(* IEC 61131-3 sources: TwinCATProj/TwinCATRD/PPS_Archive_fb/Functions/PPSFun, 11 files *)

(* ---- PPSFun.typ ---- *)
(********************************************************************
 * COPYRIGHT -- Pro Pack Systems, Inc.
 ********************************************************************
 * Library: PPSFun
 * File: PPSFun.typ
 * Author: Paul Zurlinden
 * Created: November 03, 2010
 ********************************************************************
 * Data types of library PPSFun
 ********************************************************************)

TYPE
	dtEasyLight_Outputs : 	STRUCT
		xCmdActive : BOOL;
		diResult : DINT;
		sResultText : STRING[41];
	END_STRUCT;
	dtEasyLight_InputOutput : 	STRUCT
		diCmd : DINT;
	END_STRUCT;
	dtEasyLightInterface : 	STRUCT
		Q : dtEasyLight_Outputs;
		IQ : dtEasyLight_InputOutput;
	END_STRUCT;
	dtVacCupInputs : 	STRUCT
		xEnable : BOOL;
		xEnManCntrl : BOOL;
		xManCmd : BOOL;
		tPurgeTime : TIME;
		xEmergency : BOOL;
	END_STRUCT;
	dtVacCupInputs2 : 	STRUCT
		xEnable : BOOL;
		xEnManCntrl : BOOL;
		xManCmd : BOOL;
		tPurgeTime : TIME;
		xEmergency : BOOL;
		sName : STRING[40];
		xMonitored : BOOL;
		tMonitorDelay : TIME;
	END_STRUCT;
	dtVacCup_InOut2 : 	STRUCT
		xAutoOn : BOOL;
		xAutoOff : BOOL;
		xClearFault : BOOL;
	END_STRUCT;
	dtVacCup_InOut : 	STRUCT
		xAutoOn : BOOL;
		xAutoOff : BOOL;
	END_STRUCT;
	dtVacCupOuputs : 	STRUCT
		xFBActive : BOOL;
		xSVPurge : BOOL;
		xSVVac : BOOL;
	END_STRUCT;
	dtVacCupOuputs2 : 	STRUCT
		xFBActive : BOOL;
		xSVPurge : BOOL;
		xSVVac : BOOL;
		xFault : BOOL;
		sFaultTxt : STRING[82];
	END_STRUCT;
	dtVacuumCupInterface : 	STRUCT
		I : dtVacCupInputs;
		IQ : dtVacCup_InOut;
		Q : dtVacCupOuputs;
	END_STRUCT;
	dtVacuumCupInterface2 : 	STRUCT
		I : dtVacCupInputs2;
		IQ : dtVacCup_InOut2;
		Monitor : dtDebounceInterface;
		Q : dtVacCupOuputs2;
		stErrData : dtFB_ErrorData;
	END_STRUCT;
	EnumerationEasyLight :
		(
		EN_EZL_GNSteady := 1,
		EN_EZL_RDSteady := 2,
		EN_EZL_YWSteady := 3,
		EN_EZL_BUSteady := 4,
		EN_EZL_GNFlash := 5,
		EN_EZL_RDFlash := 6,
		EN_EZL_YWFlash := 7,
		EN_EZL_BUFlash := 8,
		EN_EZL_AltGnRd := 9,
		EN_EZL_AltRdBu := 10,
		EN_EZL_AltGnYw := 11,
		EN_EZL_AltGnBu := 12,
		EN_EZL_AltRdYw := 13,
		EN_EZL_AltYwBu := 14,
		EN_EZL_AltGnRdYwBu := 15,
		EN_EZL_AllOff := 16
		);
	dtGlueApplictor : 	STRUCT
		xEnable : BOOL;
		xApplyCmd : BOOL;
		xEnManual : BOOL;
		xManPurgeCmd : BOOL;
		tPurgeTime : TIME;
		xEmergency : BOOL;
	END_STRUCT;
	dtDigCntrlInterface : 	STRUCT
		I : dtDigCntrl_Inputs;
		IQ : dtDigCntrl_InOut;
		Q : dtDigCntrl_Outputs;
		stMonitor : dtDebounceInterface;
		stErrData : dtFB_ErrorData;
	END_STRUCT;
	dtDigCntrl_Inputs : 	STRUCT
		xEnManCntrl : BOOL;
		xManCmd : BOOL;
		xEmergency : BOOL;
		xEnMonitor : BOOL;
		tMonitorDelay : TIME;
	END_STRUCT;
	dtDigCntrl_InOut : 	STRUCT
		xAutoOn : BOOL;
		xAutoOff : BOOL;
		xFaultReset : BOOL;
	END_STRUCT;
	dtDigCntrl_Outputs : 	STRUCT
		xCmd : BOOL;
		xFault : BOOL;
	END_STRUCT;
	dtFB_ErrorData : 	STRUCT
		uiErrorID : UINT;
		sErrorString : STRING[80];
		sSourceName : STRING[80];
	END_STRUCT;
	dtDebounceInterface : 	STRUCT
		I : dtDebounce_Inputs;
		Q : dtDebounce_Outputs;
	END_STRUCT;
	dtDebounce_Inputs : 	STRUCT
		xSignal : BOOL;
		tOnDelay : TIME;
		tOffDelay : TIME;
	END_STRUCT;
	dtDebounce_Outputs : 	STRUCT
		xCmd : BOOL;
		tOnTimer : TIME;
		tOffTimer : TIME;
	END_STRUCT;
	dtCylCntrlInterface : 	STRUCT
		I : dtCylCntrl_Inputs;
		IQ : dtCylCntrl_InOut;
		Q : dtCylCntrl_Outputs;
		stSensorExt : dtDebounceInterface;
		stSensorRet : dtDebounceInterface;
	END_STRUCT;
	dtCylCntrl_Inputs : 	STRUCT
		xEnableFB : BOOL;
		xValveOffRetract : BOOL;
		xAirOk : BOOL;
		xEnManCntrl : BOOL;
		xManCmd : BOOL;
		xEmergency : BOOL;
		xEnMonitor : BOOL;
		usiHWFamily : USINT;
		tTravelDel : TIME;
		xFaultReset : BOOL;
	END_STRUCT;
	dtCylCntrl_InOut : 	STRUCT
		xExtCmd : BOOL;
		xRetCmd : BOOL;
	END_STRUCT;
	dtCylCntrl_Outputs : 	STRUCT
		xFBActive : BOOL;
		xSVCmd : BOOL;
		xExtended : BOOL;
		xRetracted : BOOL;
		xFaultNoExt : BOOL;
		xFaultNoRet : BOOL;
	END_STRUCT;
END_TYPE

(* ---- FB_CylCntrl.st ---- *)
(********************************************************************
 * COPYRIGHT -- Pro Pack Systems, Inc.
 ********************************************************************
 * Library: PPSFun
 * File: FB_CylCntrl.st
 * Author: Paul Zurlinden
 * Created: November 04, 2010
 ********************************************************************
 * Implementation of library PPSFun
 ********************************************************************)

(* Controls a pneumatic cylinder with or without end of travel sensors *)
FUNCTION_BLOCK FB_CylCntrl

Timer(PT := iq_CylCntrlInterface.I.tTravelDel);
RT(CLK := iq_CylCntrlInterface.I.xManCmd);
RT_Air(CLK := iq_CylCntrlInterface.I.xAirOk);

(* Debounce Cylinder Position Sensors *)
IF iq_CylCntrlInterface.I.xEnMonitor THEN
	aFB_SensExt[0](iq_DebounceInterface := iq_CylCntrlInterface.stSensorExt);
	aFB_SensExt[1](iq_DebounceInterface := iq_CylCntrlInterface.stSensorRet);
END_IF

IF iq_CylCntrlInterface.Q.xFaultNoExt OR iq_CylCntrlInterface.Q.xFaultNoRet THEN
	xFaultSum := TRUE;
ELSE
	xFaultSum	:= FALSE;
END_IF

IF iq_CylCntrlInterface.I.xFaultReset THEN
	iq_CylCntrlInterface.Q.xFaultNoExt	:= FALSE;
	iq_CylCntrlInterface.Q.xFaultNoRet := FALSE;
END_IF

IF iq_CylCntrlInterface.I.xEnableFB THEN
	iq_CylCntrlInterface.Q.xFBActive	:= TRUE;

	(* Determine Cylinder Position when air is first turned on *)
	IF RT_Air.Q THEN
		IF iq_CylCntrlInterface.I.xEnMonitor THEN
	 		IF iq_CylCntrlInterface.stSensorExt.Q.xCmd THEN
  				iq_CylCntrlInterface.Q.xExtended		:= TRUE;
   			ELSIF iq_CylCntrlInterface.stSensorRet.Q.xCmd THEN
			 	iq_CylCntrlInterface.Q.xRetracted	:= TRUE;
   			END_IF
		ELSE
			IF iq_CylCntrlInterface.I.xValveOffRetract THEN
   				IF iq_CylCntrlInterface.Q.xSVCmd THEN
					iq_CylCntrlInterface.Q.xExtended := TRUE;
	 			ELSE
				   	iq_CylCntrlInterface.Q.xRetracted := TRUE;
	 			END_IF
			ELSE
				IF iq_CylCntrlInterface.Q.xSVCmd THEN
					iq_CylCntrlInterface.Q.xRetracted := TRUE;
	 			ELSE
				   	iq_CylCntrlInterface.Q.xExtended := TRUE;
	 			END_IF
			END_IF
		END_IF
	END_IF

	(* Fault monitor *)
	IF iq_CylCntrlInterface.I.xEnMonitor (*AND iq_CylCntrlInterface.I.usiHWFamily <> 4*) THEN (* Fault Monitor is enabled *)
		IF NOT xFaultSum THEN
			IF iq_CylCntrlInterface.I.xValveOffRetract THEN
				IF iq_CylCntrlInterface.Q.xSVCmd THEN
					IF iq_CylCntrlInterface.stSensorExt.Q.xCmd THEN
						iq_CylCntrlInterface.Q.xExtended			:= TRUE;
						iq_CylCntrlInterface.Q.xFaultNoExt		:= FALSE;
						Timer.IN												:= FALSE;
					ELSE
						IF Timer.Q THEN
							iq_CylCntrlInterface.Q.xExtended		:= FALSE;
							iq_CylCntrlInterface.Q.xFaultNoExt	:= TRUE;
							Timer.IN											:= FALSE;
						END_IF
					END_IF
				ELSE
					IF iq_CylCntrlInterface.stSensorRet.Q.xCmd THEN
						iq_CylCntrlInterface.Q.xRetracted 		:= TRUE;
						iq_CylCntrlInterface.Q.xFaultNoRet		:= FALSE;
						Timer.IN												:= FALSE;
					ELSE
						IF Timer.Q THEN
							iq_CylCntrlInterface.Q.xRetracted	:= FALSE;
							iq_CylCntrlInterface.Q.xFaultNoRet	:= TRUE;
							Timer.IN											:= FALSE;
						END_IF
					END_IF
				END_IF
			ELSE
				IF NOT iq_CylCntrlInterface.Q.xSVCmd THEN
					IF iq_CylCntrlInterface.stSensorExt.Q.xCmd THEN
						iq_CylCntrlInterface.Q.xExtended			:= TRUE;
						iq_CylCntrlInterface.Q.xFaultNoExt		:= FALSE;
						Timer.IN												:= FALSE;
					ELSE
						IF Timer.Q THEN
							iq_CylCntrlInterface.Q.xExtended		:= FALSE;
							iq_CylCntrlInterface.Q.xFaultNoExt	:= TRUE;
							Timer.IN	:= FALSE;
						END_IF
					END_IF
				ELSE
					IF iq_CylCntrlInterface.stSensorRet.Q.xCmd THEN
						iq_CylCntrlInterface.Q.xRetracted		:= TRUE;
						iq_CylCntrlInterface.Q.xFaultNoRet		:= FALSE;
						Timer.IN	:= FALSE;
					ELSE
						IF Timer.Q THEN
							iq_CylCntrlInterface.Q.xRetracted	:= FALSE;
							iq_CylCntrlInterface.Q.xFaultNoRet	:= TRUE;
							Timer.IN											:= FALSE;
						END_IF
					END_IF
				END_IF
			END_IF
		END_IF
	ELSE (* Fault Monitor is disabled *)
		IF iq_CylCntrlInterface.Q.xSVCmd THEN
			IF Timer.Q THEN
				IF iq_CylCntrlInterface.I.xValveOffRetract THEN
					iq_CylCntrlInterface.Q.xExtended		:= TRUE;
				ELSE
					iq_CylCntrlInterface.Q.xRetracted	:= TRUE;
				END_IF
				Timer.IN												:= FALSE;
			END_IF
		ELSE
			IF Timer.Q THEN
				IF iq_CylCntrlInterface.I.xValveOffRetract THEN
					iq_CylCntrlInterface.Q.xRetracted	:= TRUE;
				ELSE
					iq_CylCntrlInterface.Q.xExtended		:= TRUE;
	 			END_IF
				Timer.IN												:= FALSE;
			END_IF
		END_IF
	END_IF
	(* End Fault Monitor *)

	(* Control output *)
	IF iq_CylCntrlInterface.I.xEmergency OR xFaultSum THEN
		iq_CylCntrlInterface.Q.xSVCmd := FALSE;
	ELSE
		IF NOT iq_CylCntrlInterface.I.xEnManCntrl THEN (* When not in Manual Mode, control output *)

			IF iq_CylCntrlInterface.I.xValveOffRetract THEN
				IF iq_CylCntrlInterface.IQ.xExtCmd (*AND NOT iq_CylCntrlInterface.Q.xSVCmd*) THEN
					iq_CylCntrlInterface.Q.xSVCmd		:= TRUE;
					iq_CylCntrlInterface.Q.xRetracted	:= FALSE;
					iq_CylCntrlInterface.Q.xExtended		:= FALSE;
					Timer.IN											:= TRUE;
					IF iq_CylCntrlInterface.Q.xSVCmd THEN
						iq_CylCntrlInterface.IQ.xExtCmd		:= FALSE;
					END_IF
				END_IF

				IF iq_CylCntrlInterface.IQ.xRetCmd (*AND iq_CylCntrlInterface.Q.xSVCmd*) THEN
					iq_CylCntrlInterface.Q.xSVCmd		:= FALSE;
					iq_CylCntrlInterface.Q.xExtended		:= FALSE;
					iq_CylCntrlInterface.Q.xRetracted	:= FALSE;
					Timer.IN											:= TRUE;
					IF NOT iq_CylCntrlInterface.Q.xSVCmd THEN
						iq_CylCntrlInterface.IQ.xRetCmd		:= FALSE;
					END_IF
				END_IF
			ELSE
				IF iq_CylCntrlInterface.IQ.xExtCmd (*AND iq_CylCntrlInterface.Q.xSVCmd*) THEN
					iq_CylCntrlInterface.Q.xSVCmd		:= FALSE;
					iq_CylCntrlInterface.Q.xExtended		:= FALSE;
					iq_CylCntrlInterface.Q.xRetracted	:= FALSE;
					Timer.IN											:= TRUE;
					IF NOT iq_CylCntrlInterface.Q.xSVCmd THEN
						iq_CylCntrlInterface.IQ.xExtCmd		:= FALSE;
					END_IF
				END_IF

				IF iq_CylCntrlInterface.IQ.xRetCmd (*AND NOT iq_CylCntrlInterface.Q.xSVCmd*) THEN
					iq_CylCntrlInterface.Q.xSVCmd		:= TRUE;
					iq_CylCntrlInterface.Q.xExtended		:= FALSE;
					iq_CylCntrlInterface.Q.xRetracted	:= FALSE;
					Timer.IN											:= TRUE;
					IF iq_CylCntrlInterface.Q.xSVCmd THEN
						iq_CylCntrlInterface.IQ.xRetCmd		:= FALSE;
					END_IF
				END_IF
			END_IF

		ELSE (* When in Manual Mode, control output *)
			IF iq_CylCntrlInterface.Q.xSVCmd THEN
				IF RT.Q THEN
					iq_CylCntrlInterface.Q.xSVCmd		:= FALSE;
					iq_CylCntrlInterface.Q.xRetracted	:= FALSE;
					iq_CylCntrlInterface.Q.xExtended		:= FALSE;
					Timer.IN											:= TRUE;
				END_IF
			ELSE
				IF RT.Q THEN
					iq_CylCntrlInterface.Q.xSVCmd		:= TRUE;
					iq_CylCntrlInterface.Q.xRetracted	:= FALSE;
					iq_CylCntrlInterface.Q.xExtended		:= FALSE;
					Timer.IN											:= TRUE;
				END_IF
			END_IF
		END_IF
	END_IF

ELSE
	iq_CylCntrlInterface.Q.xFBActive		:= FALSE;
	iq_CylCntrlInterface.Q.xSVCmd		:= FALSE;
	iq_CylCntrlInterface.Q.xExtended		:= FALSE;
	iq_CylCntrlInterface.Q.xRetracted	:= FALSE;
	Timer.IN	:= FALSE;
END_IF

END_FUNCTION_BLOCK

(* ---- FB_Debounce.st ---- *)
(********************************************************************
 * COPYRIGHT -- Pro Pack Systems, Inc.
 ********************************************************************
 * Library: PPSFun
 * File: FB_Debounce.st
 * Author: Paul Zurlinden
 * Created: November 03, 2010
 ********************************************************************
 * Implementation of library PPSFun
 ********************************************************************)

(* Filter an input with On and Off delays *)
FUNCTION_BLOCK FB_Debounce

tmrOn(IN := iq_DebounceInterface.I.xSignal, PT := iq_DebounceInterface.I.tOnDelay);
tmrOff(IN := tmrOn.Q, PT := iq_DebounceInterface.I.tOffDelay);

iq_DebounceInterface.Q.xCmd			:= tmrOff.Q;
iq_DebounceInterface.Q.tOnTimer		:= tmrOn.ET;
iq_DebounceInterface.Q.tOffTimer		:= tmrOff.ET;

END_FUNCTION_BLOCK

(* ---- FB_DigCntrl.st ---- *)
(********************************************************************
 * COPYRIGHT -- Pro Pack Systems, Inc.
 ********************************************************************
 * Library: PPSFun
 * File: FB_DigCntrl.st
 * Author: Paul Zurlinden
 * Created: May 26, 2011
 ********************************************************************
 * Implementation of library PPSFun
 ********************************************************************)

(* Controls a digital output in the following ways;

		**** Must use dtDigCntrlInterface with this FB ****

		Allows a manual mode for only a momentary manual cmd to toggle the output
		If not in manual mode, allows for xAutoOn to be high to toggle output On,
			Conversly, allows xAutoOff to be high to toggle output Off.  xAutoOn and xAutoOff
			are set low by FB when scanned.
		Also if xEnMonitor is true monitors output with an input xMonitor in conjuction with a
			delay timer tMonitorDelay such that if the output is on, the monitor input must be high
			within the time specified by the delay else a fault is triggered which disables the output
			or any command to toggle it.*)

FUNCTION_BLOCK FB_DigCntrl

RT(CLK := iq_DigCntrlInterface.I.xManCmd);

IF iq_DigCntrlInterface.I.xEnMonitor THEN
	FB_MonitorDebounce(iq_DebounceInterface := iq_DigCntrlInterface.stMonitor);
END_IF

IF iq_DigCntrlInterface.I.xEmergency THEN
	iq_DigCntrlInterface.Q.xCmd := FALSE;
END_IF

IF NOT iq_DigCntrlInterface.Q.xFault AND NOT iq_DigCntrlInterface.I.xEmergency THEN
	IF iq_DigCntrlInterface.I.xEnManCntrl THEN
		IF RT.Q THEN
	 		IF iq_DigCntrlInterface.Q.xCmd THEN
  				iq_DigCntrlInterface.Q.xCmd := FALSE;
  	 		ELSE
			 	iq_DigCntrlInterface.Q.xCmd := TRUE;
	   		END_IF
		END_IF
	ELSE
//		IF iq_DigCntrlInterface.Q.xCmd THEN
	 		IF iq_DigCntrlInterface.IQ.xAutoOff THEN
	  			iq_DigCntrlInterface.Q.xCmd		:= FALSE;
				iq_DigCntrlInterface.IQ.xAutoOff	:= FALSE;
	   		END_IF
//		ELSE
			IF iq_DigCntrlInterface.IQ.xAutoOn THEN
	  			iq_DigCntrlInterface.Q.xCmd		:= TRUE;
				iq_DigCntrlInterface.IQ.xAutoOn	:= FALSE;
	   		END_IF
//		END_IF
	END_IF
END_IF

IF iq_DigCntrlInterface.I.xEnMonitor (*AND iq_DigCntrlInterface.I.usiHWFamily <> 4*) THEN
	Timer(IN := iq_DigCntrlInterface.Q.xCmd, PT := iq_DigCntrlInterface.I.tMonitorDelay);

	IF Timer.Q AND NOT iq_DigCntrlInterface.stMonitor.Q.xCmd THEN
		iq_DigCntrlInterface.Q.xFault	:= TRUE;
		iq_DigCntrlInterface.Q.xCmd	:= FALSE;
	END_IF

	IF iq_DigCntrlInterface.IQ.xFaultReset THEN
		iq_DigCntrlInterface.Q.xFault 		:= FALSE;
		iq_DigCntrlInterface.IQ.xFaultReset	:= FALSE;
	END_IF
END_IF

END_FUNCTION_BLOCK

(* ---- FB_EZLight.st ---- *)
(********************************************************************
 * COPYRIGHT -- Pro Pack Systems, Inc.
 ********************************************************************
 * Library: PPSFun
 * File: FB_EZLight.st
 * Author: Paul Zurlinden
 * Created: November 05, 2010
 ********************************************************************
 * Implementation of library PPSFun
 ********************************************************************)

(* Controls Banner Light K50LGRYB4PQ *)
FUNCTION_BLOCK FB_EZLight

IF iq_diCmd <> 0 THEN
	q_diResult := iq_diCmd;
	IF iq_diCmd = q_diResult THEN
		iq_diCmd :=0;
	END_IF
END_IF

IF q_xGnLight OR q_xRdLight OR q_xYwLight OR q_xBuLight THEN
	q_xLightActive := TRUE;
ELSE
	q_xLightActive := FALSE;
END_IF

CASE q_diResult OF

	EN_EZL_GNSteady:
		q_xGnLight := TRUE;
		q_xRdLight	:= FALSE;
  		q_xBuLight	:= FALSE;
  		q_xYwLight	:= FALSE;
		q_sResultText := 'Green Steady';

	EN_EZL_GNFlash:
		q_xGnLight := TRUE;
		q_xYwLight := TRUE;
		q_xBuLight	:= FALSE;
  		q_xRdLight	:= FALSE;
		q_sResultText := 'Green Flashing';

	EN_EZL_RDSteady:
		q_xRdLight := TRUE;
		q_xGnLight	:= FALSE;
  		q_xYwLight	:= FALSE;
  		q_xBuLight	:= FALSE;
		q_sResultText := 'Red Steady';

	EN_EZL_RDFlash:
		q_xRdLight := TRUE;
		q_xGnLight := TRUE;
		q_xYwLight	:= FALSE;
  		q_xBuLight	:= FALSE;
		q_sResultText := 'Red Flashing';

	EN_EZL_YWSteady:
		q_xYwLight := TRUE;
		q_xGnLight	:= FALSE;
  		q_xRdLight	:= FALSE;
  		q_xBuLight	:= FALSE;
		q_sResultText := 'Yellow Steady';

	EN_EZL_YWFlash:
		q_xYwLight :=TRUE;
		q_xRdLight := TRUE;
		q_xBuLight	:= FALSE;
  		q_xGnLight	:= FALSE;
		q_sResultText := 'Yellow Flashing';

	EN_EZL_BUSteady:
		q_xBuLight := TRUE;
		q_xGnLight	:= FALSE;
  		q_xRdLight	:= FALSE;
  		q_xYwLight	:= FALSE;
		q_sResultText := 'Blue Steady';

	EN_EZL_BUFlash:
		q_xBuLight := TRUE;
		q_xRdLight := TRUE;
		q_xYwLight	:= FALSE;
  		q_xGnLight	:= FALSE;
		q_sResultText := 'Blue Flashing';

	EN_EZL_AltGnRd:
		q_xGnLight := TRUE;
		q_xBuLight := TRUE;
		q_xYwLight	:= FALSE;
  		q_xRdLight	:= FALSE;
		q_sResultText := 'Alternating Green and Red';

	EN_EZL_AltRdBu:
		q_xYwLight := TRUE;
		q_xBuLight := TRUE;
		q_xGnLight	:= FALSE;
  		q_xRdLight	:= FALSE;
		q_sResultText := 'Alternating Red and Blue';

	EN_EZL_AltGnYw:
		q_xGnLight := TRUE;
		q_xYwLight := TRUE;
		q_xBuLight := TRUE;
		q_xRdLight	:= FALSE;
		q_sResultText := 'Alternating Green and Yellow';

	EN_EZL_AltGnBu:
		q_xGnLight := TRUE;
		q_xRdLight := TRUE;
		q_xBuLight := TRUE;
		q_xYwLight	:= FALSE;
		q_sResultText := 'Alternating Green and Blue';

	EN_EZL_AltRdYw:
		q_xRdLight := TRUE;
		q_xYwLight := TRUE;
		q_xBuLight := TRUE;
		q_xGnLight	:= FALSE;
		q_sResultText := 'Alternating Red and Yellow';

	EN_EZL_AltYwBu:
		q_xGnLight := TRUE;
		q_xRdLight := TRUE;
		q_xYwLight := TRUE;
		q_xBuLight	:= FALSE;
		q_sResultText := 'Alternating Yellow and Blue';

	EN_EZL_AltGnRdYwBu:
		q_xGnLight := TRUE;
		q_xRdLight := TRUE;
		q_xYwLight := TRUE;
		q_xBuLight := TRUE;
		q_sResultText := 'Alternating Green, Red, Yellow and Blue';

	EN_EZL_AllOff:
		q_xGnLight := FALSE;
		q_xRdLight := FALSE;
		q_xYwLight := FALSE;
		q_xBuLight := FALSE;
		q_sResultText := 'All Off';

END_CASE

END_FUNCTION_BLOCK

(* ---- FB_Flasher.st ---- *)
(********************************************************************
 * COPYRIGHT -- Pro Pack Systems, Inc.
 ********************************************************************
 * Library: PPSFun
 * File: FB_Flasher.st
 * Author: PaulZ
 * Created: December 29, 2010
 ********************************************************************
 * Implementation of library PPSFun
 ********************************************************************)

(* Flasher *)
FUNCTION_BLOCK FB_Flasher

tmrOn(PT := i_tOn);
tmrOff(IN := tmrOn.Q, PT := i_tOff);

IF i_xSignal AND NOT tmrOff.Q THEN
	tmrOn.IN	:= TRUE;
ELSE
	tmrOn.IN	:= FALSE;
END_IF

q_xFlash	:= tmrOff.Q;

END_FUNCTION_BLOCK

(* ---- FB_GlueApplicator.st ---- *)
(********************************************************************
 * COPYRIGHT -- Pro Pack Systems, Inc.
 ********************************************************************
 * Library: PPSFun
 * File: FB_GlueApplicator.st
 * Author: Paul Zurlinden
 * Created: November 05, 2010
 ********************************************************************
 * Implementation of library PPSFun
 ********************************************************************)

(* Controls Glue Applicator for Auto and Manual Mode *)
FUNCTION_BLOCK FB_GlueApplicator

RT(CLK := i_xManPurgeCmd);

Timer(PT := i_tPurgeTime);
IF Timer.Q THEN
	Timer.IN := FALSE;
END_IF

IF i_xEnable THEN

	IF i_xEnManual AND RT.Q THEN
 		Timer.IN := TRUE;
  	END_IF

	IF Timer.IN OR i_xApplyCmd THEN
 		q_xApplicatorEnable := TRUE;
  	ELSE
		q_xApplicatorEnable := FALSE;
  	END_IF

ELSIF i_xEmergency OR NOT i_xEnable THEN

	q_xApplicatorEnable := FALSE;
 	Timer.IN := FALSE;

END_IF

END_FUNCTION_BLOCK

(* ---- FB_Toggle.st ---- *)
(********************************************************************
 * COPYRIGHT -- Pro Pack Systems, Inc.
 ********************************************************************
 * Library: PPSFun
 * File: FB_Toggle.st
 * Author: Paul Zurlinden
 * Created: November 04, 2010
 ********************************************************************
 * Implementation of library PPSFun
 ********************************************************************)

(* Monitors momentary input and toggles the output *)
FUNCTION_BLOCK FB_Toggle

counter(
	CU := i_xMomentary,
	RESET := i_xEmergency);

q_xCMD := counter.Q;

END_FUNCTION_BLOCK

(* ---- FB_VacCup.st ---- *)
(********************************************************************
 * COPYRIGHT -- Pro Pack Systems, Inc.
 ********************************************************************
 * Library: PPSFun
 * File: FB_VacCup.st
 * Author: Paul Zurlinden
 * Created: November 09, 2010
 ********************************************************************
 * Implementation of library PPSFun
 ********************************************************************)

(* Controls a vacuum cup with purge *)
FUNCTION_BLOCK FB_VacCup
RT(CLK := iq_VacCupInterface.I.xManCmd);
FT(CLK := iq_VacCupInterface.Q.xSVVac);
Timer(PT := iq_VacCupInterface.I.tPurgeTime);

IF iq_VacCupInterface.I.xEnable AND NOT iq_VacCupInterface.I.xEmergency THEN
	iq_VacCupInterface.Q.xFBActive	:= TRUE;
	(* Control the vacuum valve *)
	IF iq_VacCupInterface.I.xEnManCntrl THEN
		IF RT.Q THEN
	 		IF iq_VacCupInterface.Q.xSVVac THEN
  				iq_VacCupInterface.Q.xSVVac := FALSE;
  	 		ELSE
			 	iq_VacCupInterface.Q.xSVVac := TRUE;
	   		END_IF
		END_IF
	ELSE
//		IF iq_VacCupInterface.Q.xSVVac THEN
	 		IF iq_VacCupInterface.IQ.xAutoOff THEN
	  			iq_VacCupInterface.Q.xSVVac	:= FALSE;
				iq_VacCupInterface.IQ.xAutoOff	:= FALSE;
	   		END_IF
//		ELSE
			IF iq_VacCupInterface.IQ.xAutoOn THEN
	  			iq_VacCupInterface.Q.xSVVac	:= TRUE;
				iq_VacCupInterface.IQ.xAutoOn	:= FALSE;
	   		END_IF
		END_IF
//	END_IF

	(* Control the purge valve *)
	IF FT.Q THEN
 		Timer.IN 		:= TRUE;
  	END_IF

	IF Timer.Q THEN
 		Timer.IN		:= FALSE;
  	END_IF

	iq_VacCupInterface.Q.xSVPurge		:= Timer.IN;

ELSIF iq_VacCupInterface.I.xEmergency THEN
	Timer.IN		:= FALSE;
 	iq_VacCupInterface.Q.xSVVac		:= FALSE;
 	iq_VacCupInterface.Q.xSVPurge		:= FALSE;
ELSIF NOT iq_VacCupInterface.I.xEnable THEN
	Timer.IN		:= FALSE;
 	iq_VacCupInterface.Q.xSVVac		:= FALSE;
 	iq_VacCupInterface.Q.xSVPurge		:= FALSE;
	iq_VacCupInterface.Q.xFBActive	:= FALSE;
END_IF

END_FUNCTION_BLOCK

(* ---- FB_VacCup2.st ---- *)
(********************************************************************
 * COPYRIGHT -- Pro Pack Systems, Inc.
 ********************************************************************
 * Library: PPSFun
 * File: FB_VacCup2.st
 * Author: PaulZ
 * Created: March 19, 2013
 ********************************************************************
 * Implementation of library PPSFun
 ********************************************************************)

(* Controls seperate valves for vacuum and purge, impliments a monitoring input. *)
FUNCTION_BLOCK FB_VacCup2

	RT(CLK := iq_VacCupInterface.I.xManCmd);
	FT(CLK := iq_VacCupInterface.Q.xSVVac);
	Timer(PT := iq_VacCupInterface.I.tPurgeTime);
	tmrMon(PT := iq_VacCupInterface.I.tMonitorDelay);
	ifbMonitor(iq_DebounceInterface := iq_VacCupInterface.Monitor);

	IF iq_VacCupInterface.Q.xFault THEN
		iq_VacCupInterface.Q.xSVVac	:= FALSE;
		iq_VacCupInterface.IQ.xAutoOff	:= FALSE;
		iq_VacCupInterface.IQ.xAutoOn	:= FALSE;
	END_IF

	IF (tmrMon.Q) AND (NOT xHadVac) THEN
		tmrMon.IN								:= FALSE;
		iq_VacCupInterface.Q.xFault	:= TRUE;
  		iq_VacCupInterface.Q.sFaultTxt	:= CONCAT(iq_VacCupInterface.I.sName, ' could not vacuum');
	END_IF

	IF iq_VacCupInterface.Q.xFault AND iq_VacCupInterface.IQ.xClearFault THEN
 		iq_VacCupInterface.Q.xFault			:= FALSE;
		iq_VacCupInterface.Q.sFaultTxt		:= '';
		xHadVac								:= FALSE;
		iq_VacCupInterface.IQ.xClearFault	:= FALSE;
	END_IF

	IF iq_VacCupInterface.I.xEnable AND NOT iq_VacCupInterface.I.xEmergency THEN

		iq_VacCupInterface.Q.xFBActive	:= TRUE;

		(* Control the vacuum valve *)
		IF iq_VacCupInterface.I.xEnManCntrl THEN
			iq_VacCupInterface.IQ.xAutoOff	:= FALSE;
			iq_VacCupInterface.IQ.xAutoOn	:= FALSE;
			IF RT.Q THEN
		 		IF iq_VacCupInterface.Q.xSVVac THEN
	  				iq_VacCupInterface.Q.xSVVac := FALSE;
	  	 		ELSE
				 	iq_VacCupInterface.Q.xSVVac := TRUE;
		   		END_IF
			END_IF
		ELSE

		 	IF iq_VacCupInterface.IQ.xAutoOff THEN
		  		iq_VacCupInterface.Q.xSVVac	:= FALSE;
				iq_VacCupInterface.IQ.xAutoOff	:= FALSE;
				IF iq_VacCupInterface.I.xMonitored THEN
					tmrMon.IN									:= FALSE;
				END_IF
				xHadVac										:= FALSE;
		  	END_IF

			IF iq_VacCupInterface.IQ.xAutoOn THEN
		  		iq_VacCupInterface.Q.xSVVac	:= TRUE;
				iq_VacCupInterface.IQ.xAutoOn	:= FALSE;
				IF iq_VacCupInterface.I.xMonitored THEN
					tmrMon.IN									:= TRUE;
				END_IF
		  	END_IF

		END_IF

		(* Monitor for Vacuum *)
		IF	(iq_VacCupInterface.I.xMonitored)
			AND (iq_VacCupInterface.Q.xSVVac)
			AND (NOT tmrMon.Q)
			AND iq_VacCupInterface.Monitor.Q.xCmd THEN
				xHadVac		:= TRUE;
  				tmrMon.IN	:= FALSE;
  		END_IF

		IF (iq_VacCupInterface.I.xMonitored)
			AND (NOT iq_VacCupInterface.I.xEnManCntrl)
   			AND (iq_VacCupInterface.Q.xSVVac)
   			AND (xHadVac)
			AND (NOT iq_VacCupInterface.Monitor.Q.xCmd) THEN
   				iq_VacCupInterface.Q.xFault	:= TRUE;
				iq_VacCupInterface.Q.sFaultTxt := CONCAT(iq_VacCupInterface.I.sName, ' lost vacuum');
		END_IF

		(* Control the purge valve *)
		IF (FT.Q) AND (NOT iq_VacCupInterface.Q.xFault) THEN
	 		Timer.IN 		:= TRUE;
	  	END_IF

		IF Timer.Q THEN
	 		Timer.IN		:= FALSE;
	  	END_IF

		iq_VacCupInterface.Q.xSVPurge		:= Timer.IN;

	ELSIF iq_VacCupInterface.I.xEmergency THEN
		Timer.IN										:= FALSE;
	 	iq_VacCupInterface.Q.xSVVac		:= FALSE;
	 	iq_VacCupInterface.Q.xSVPurge		:= FALSE;
	ELSIF NOT iq_VacCupInterface.I.xEnable THEN
		Timer.IN										:= FALSE;
	 	iq_VacCupInterface.Q.xSVVac		:= FALSE;
	 	iq_VacCupInterface.Q.xSVPurge		:= FALSE;
		iq_VacCupInterface.Q.xFBActive		:= FALSE;
		iq_VacCupInterface.Q.xFault			:= FALSE;
  		iq_VacCupInterface.Q.sFaultTxt		:= '';
	END_IF

END_FUNCTION_BLOCK

(* ---- PPSFun.fun ---- *)
(********************************************************************
 * COPYRIGHT -- Pro Pack Systems, Inc.
 ********************************************************************
 * Library: PPSFun
 * File: PPSFun.fun
 * Author: Paul Zurlinden
 * Created: November 03, 2010
 ********************************************************************
 * Functions and function blocks of library PPSFun
 ********************************************************************)

FUNCTION_BLOCK FB_Debounce (*Filter an input with On and Off delays*)
	VAR_IN_OUT
		iq_DebounceInterface : dtDebounceInterface;
	END_VAR
	VAR
		tmrOn : TON;
		tmrOff : TOF;
	END_VAR
END_FUNCTION_BLOCK

FUNCTION_BLOCK FB_Toggle (*Monitors momentary input and toggles the output*)
	VAR_INPUT
		i_xMomentary : BOOL;
		i_xEmergency : BOOL;
	END_VAR
	VAR_OUTPUT
		q_xCMD : BOOL;
	END_VAR
	VAR
		counter : CTU;
	END_VAR
END_FUNCTION_BLOCK

FUNCTION_BLOCK FB_DigCntrl
	VAR_IN_OUT
		iq_DigCntrlInterface : dtDigCntrlInterface;
	END_VAR
	VAR
		RT : R_TRIG;
		Timer : TON;
		FB_MonitorDebounce : FB_Debounce;
	END_VAR
END_FUNCTION_BLOCK

FUNCTION_BLOCK FB_CylCntrl (*Controls a pneumatic cylinder with or without end of travel sensors*)
	VAR_IN_OUT
		iq_CylCntrlInterface : dtCylCntrlInterface;
	END_VAR
	VAR
		RT : R_TRIG;
		Timer : TON;
		RT_Air : R_TRIG;
		xFaultSum : BOOL;
		aFB_SensExt : ARRAY[0..1] OF FB_Debounce;
	END_VAR
END_FUNCTION_BLOCK

FUNCTION_BLOCK FB_EZLight (*Controls Banner Light K50LGRYB4PQ*)
	VAR_OUTPUT
		q_xCmdActive : BOOL;
		q_diResult : DINT;
		q_sResultText : STRING[41];
		q_xLightActive : BOOL;
		q_xGnLight : BOOL;
		q_xRdLight : BOOL;
		q_xYwLight : BOOL;
		q_xBuLight : BOOL;
	END_VAR
	VAR_IN_OUT
		iq_diCmd : DINT;
	END_VAR
END_FUNCTION_BLOCK

FUNCTION_BLOCK FB_GlueApplicator (*Controls Glue Applicator for Auto and Manual Mode*)
	VAR_INPUT
		i_xEnable : BOOL;
		i_xApplyCmd : BOOL;
		i_xEnManual : BOOL;
		i_xManPurgeCmd : BOOL;
		i_tPurgeTime : TIME;
		i_xEmergency : BOOL;
	END_VAR
	VAR_OUTPUT
		q_xApplicatorEnable : BOOL;
	END_VAR
	VAR
		RT : R_TRIG;
		Timer : TON;
	END_VAR
END_FUNCTION_BLOCK

FUNCTION_BLOCK FB_VacCup (*Controls a vacuum cup with purge*)
	VAR_IN_OUT
		iq_VacCupInterface : dtVacuumCupInterface;
	END_VAR
	VAR
		Timer : TON;
		RT : R_TRIG;
		FT : F_TRIG;
	END_VAR
END_FUNCTION_BLOCK

FUNCTION_BLOCK FB_Flasher (*Flasher*)
	VAR_INPUT
		i_xSignal : BOOL;
		i_tOn : TIME;
		i_tOff : TIME;
	END_VAR
	VAR_OUTPUT
		q_xFlash : BOOL;
	END_VAR
	VAR
		tmrOn : TON;
		tmrOff : TOF;
	END_VAR
END_FUNCTION_BLOCK

FUNCTION_BLOCK FB_VacCup2 (*Controls seperate valves for vacuum and purge, impliments a monitoring input.*)
	VAR_IN_OUT
		iq_VacCupInterface : dtVacuumCupInterface2;
	END_VAR
	VAR
		Timer : TON;
		RT : R_TRIG;
		FT : F_TRIG;
		tmrMon : TON;
		ifbMonitor : FB_Debounce;
		xHadVac : BOOL;
	END_VAR
END_FUNCTION_BLOCK
